// TIA Portal V20 export
DATA_BLOCK "Config"   // DB42
{ DB_Accessible_From_OPC_UA := 'FALSE' }
AUTHOR : ERsystem_FA2_DH. Kim
// stored: Access Published, DBAccessibleFromOPCUA false, DBAccessibleFromWebserver false, MemoryReserve 100, Namespace Unit1.Em1
   VAR RETAIN
      em { ExternalWritable := 'False'} : "LAF_typeEmConfiguration";
      axis { ExternalAccessible := 'False'; ExternalVisible := 'False'; ExternalWritable := 'False'} : Array[1.._.U1EM1_NO_OF_AXES] of DB_ANY;
      cmUnwinderBtmAxisB { ExternalAccessible := 'False'; ExternalVisible := 'False'; ExternalWritable := 'False'} : "LBC_typeAxis64PosConfiguration";
      cmAirShaftBtmOnOff { ExternalAccessible := 'False'; ExternalVisible := 'False'; ExternalWritable := 'False'} : "LBC_typeTwoWayActuatorConfiguration";
      cmRadiusMeasureBtm { ExternalAccessible := 'False'; ExternalVisible := 'False'; ExternalWritable := 'False'} : "LBC_typeAnalogInputConfiguration";
      cmEpcBtm { ExternalAccessible := 'False'; ExternalVisible := 'False'; ExternalWritable := 'False'} : "LER_typeCON600Configuration";
      cmBtmDirectionCheckSensor { S7_SetPoint := 'True'} : "LBC_typeDigitalSignalConfiguration";
      cmRadiusMeasure : "LER_typeRadiusMeasureConfiguration";
      softCam : Struct
         unwinderBtmAxisB : "LER_typeSoftCamInterface";
      END_STRUCT;
      Data : Array[0..10] of LReal;
   END_VAR
BEGIN
   em.referenceDesignator.parent := WSTRING#'U1';
   em.referenceDesignator.relative := WSTRING#'EM1 SepaUnwinderBtm';
   em.referenceDesignator.combined := WSTRING#'U1.EM1 SepaUnwinderBtm';
   axis[1] := 85;
   axis[2] := 263;
   cmUnwinderBtmAxisB.referenceDesignator := WSTRING#'cmUnwinderBtmAxisB';
   cmAirShaftBtmOnOff.referenceDesignator := WSTRING#'cmAirShaftBtmOnOff';
   cmAirShaftBtmOnOff.monitoringLeavingFeedback := T#500ms;
   cmAirShaftBtmOnOff.monitoringReachingFeedback := T#500ms;
   cmAirShaftBtmOnOff.monitoringDiscrepancy := T#0MS;
   cmAirShaftBtmOnOff.setOutputHomeContinuously := TRUE;
   cmAirShaftBtmOnOff.setOutputWorkContinuously := TRUE;
   cmAirShaftBtmOnOff.disableHomeCommand := FALSE;
   cmAirShaftBtmOnOff.disableFeedbackHomePos := FALSE;
   cmAirShaftBtmOnOff.disableFeedbackWorkPos := FALSE;
   cmAirShaftBtmOnOff.disableAlarms := FALSE;
   cmAirShaftBtmOnOff.resetOutputsOnError := FALSE;
   cmAirShaftBtmOnOff.allwaysWaitOnReachingTime := FALSE;
   cmRadiusMeasureBtm.referenceDesignator := WSTRING#'cmRadiusMeasureBtm';
   cmRadiusMeasureBtm.physicalUnit := 'unit';
   cmRadiusMeasureBtm.isUnipolarSignal := TRUE;
   cmRadiusMeasureBtm.default := 0.0;
   cmRadiusMeasureBtm.limitHigh2 := 400.0;
   cmRadiusMeasureBtm.limitHigh1 := 400.0;
   cmRadiusMeasureBtm.limitLow1 := 0.0;
   cmRadiusMeasureBtm.limitLow2 := 0.0;
   cmRadiusMeasureBtm.processValueMax := 400.0;
   cmRadiusMeasureBtm.processValueMin := 0.0;
   cmRadiusMeasureBtm.scaleAnalogUppPoint := 27648.0;
   cmRadiusMeasureBtm.scaleAnalogLowPoint := 0.0;
   cmRadiusMeasureBtm.scaleProcessUppPoint := 400.0;
   cmRadiusMeasureBtm.scaleProcessLowPoint := 0.0;
   cmRadiusMeasureBtm.disableAlarms := TRUE;
   cmBtmDirectionCheckSensor.referenceDesignator := WSTRING#'cmBtmDirectionCheckSensor';
   cmBtmDirectionCheckSensor.onDelay := T#0MS;
   cmBtmDirectionCheckSensor.offDelay := T#0MS;
   cmBtmDirectionCheckSensor.default := FALSE;
   cmBtmDirectionCheckSensor.invertProcessValue := FALSE;
   cmBtmDirectionCheckSensor.disableAlarms := FALSE;
   cmRadiusMeasure.Offset := 39.0;
   cmRadiusMeasure.DecimalPoint := 1;
END_DATA_BLOCK
